INTERFACE I_Mc3MotionPowerTask EXTENDS I_Mc2MotionTask, I_AxisEnable

END_INTERFACE

(* stored: Version 1.1.0.1, ProductVersion 3.1.4026.20
   Itf I_Mc3MotionPowerTask: Id {dc7d1f9a-718d-4cce-a7ad-66e6fbe71707} *)
